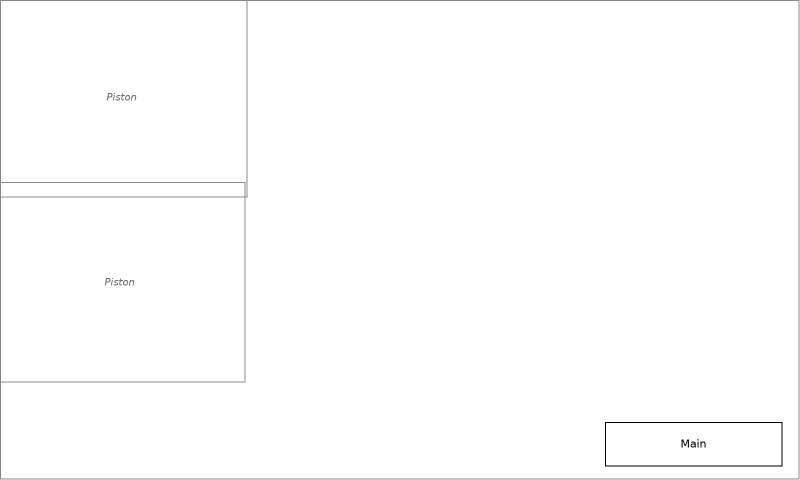
VISUALIZATION GripperManual  // 800x480
    Frame (-3,-3 250x200)
        shows Piston(piston := GVL_HMI.stGripSolL)
    Rectangle (605,422 177x44), "Main"
        OnMouseDown: change screen: Main
    Frame (-5,182 250x200)
        shows Piston(piston := GVL_HMI.stGripSolR)
END_VISUALIZATION

(* stored: Version 1.1.0.1, ProductVersion 3.1.4024.16
   Visu GripperManual: Id {a1b2c3d4-0e5f-4a6b-9c7d-000000000101} *)
